{attribute 'qualified_only'}
VAR_GLOBAL
END_VAR

(* stored: Version 1.1.0.1, ProductVersion 3.1.4024.16
   GVL Global: Id {4b021af1-77a6-4279-b1dd-bdd9bb666e7c} *)
